// SIMATIC S7-200 project (STEP 7-Micro/WIN), CPU 222 REL 01.22

SYMBOL_TABLE USUARIO1
FR1              I0.0     // RELE TERMICO
S1               I0.1     // PULSADOR PARO
S2               I0.2     // PULSADOR DE MARCHA
KM1              Q0.0     // CONTACTOR MOTOR1
KM2              Q0.1     // CONTACTOR MOTOR2
KM3              Q0.2     // CONTACTOR MOTOR3
H1               Q0.3     // SEÑALIZACION AVERIA
END_SYMBOL_TABLE

ORGANIZATION_BLOCK PRINCIPAL:OB1
TITLE=COMENTARIOS DEL PROGRAMA
BEGIN
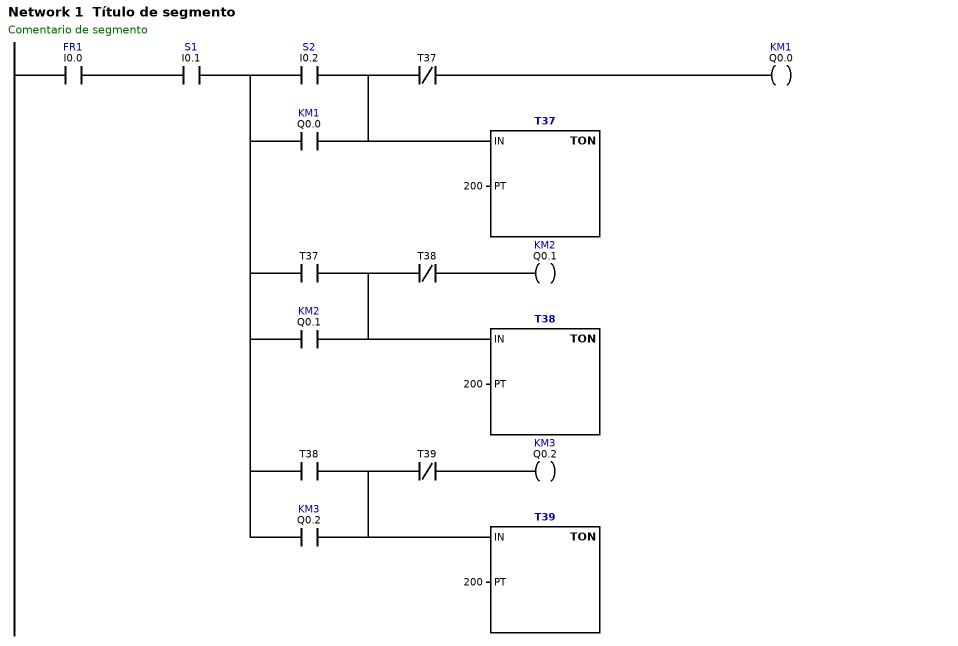
Network 1 // Título de segmento
// Comentario de segmento
// (network saved uncompiled; LAD cells follow)
// row 0: c0 -| |- FR1:I0.0  c1 -| |- S1:I0.1 v  c2 -| |- S2:I0.2 v  c3 -|/|- T37  c4 --  c5 --  c6 -( ) KM1:Q0.0
// row 1: c1 ^v  c2 -| |- KM1:Q0.0 ^  c3 --  c4 [TON T37 IN:=power@row1, PT:=200]
// row 2: c1 ^v  c4 [box]
// row 3: c1 ^v  c2 -| |- T37 v  c3 -|/|- T38  c4 -( ) KM2:Q0.1
// row 4: c1 ^v  c2 -| |- KM2:Q0.1 ^  c3 --  c4 [TON T38 IN:=power@row4, PT:=200]
// row 5: c1 ^v  c4 [box]
// row 6: c1 ^v  c2 -| |- T38 v  c3 -|/|- T39  c4 -( ) KM3:Q0.2
// row 7: c1 ^  c2 -| |- KM3:Q0.2 ^  c3 --  c4 [TON T39 IN:=power@row7, PT:=200]
// row 8: c4 [box]
END_ORGANIZATION_BLOCK
